{attribute 'qualified_only'}
VAR_GLOBAL
	//Lista of single structure variables
	rParameter01 : Parameter;
	rParameter02 : Parameter;
	rParameter03 : Parameter;
	rParameter04 : Parameter;
	rParameter05 : Parameter;
	rParameter06 : Parameter;
	rParameter07 : Parameter;
	rParameter08 : Parameter;
	
	//Array of structure
	aParameters : ARRAY [0..9] OF Parameter;
END_VAR

(* stored: Version 1.1.0.1, ProductVersion 3.1.4024.4
   GVL Parameters: Id {29f0d58c-14cb-49f4-9e0b-3c230de6166c} *)
